(* Logix 5000 project; controller Carpenter_Meter_SCP vendor 1 type 14 code 217 rev 31.11; software revision 31.01 *)

TASK MainTask (continuous, watchdog 500 ms) : First_Scan, Map_Inputs, Alarm_Shutdown, Valve_Control, Station_Overrides, Station_Control, Meter_Skid_Control, Auxiliary_Control, Communication, Map_Outputs, OCC_Comms

MODULES
   Local : vendor 1 type 14 code 217 (5069 0, rev 31.11)
      Carpenter_Meter_FGP : vendor 1 type 14 code 217 (Ethernet 10.131.51.170, rev 31.1, $eaa37dee$ RPI 20 ms, $a3d2e279$ RPI 20 ms)
      MLV_HRF100 : vendor 1 type 14 code 107 (Ethernet 10.171.255.104, rev 31.1)
      Hereford_Meter_SCP : vendor 1 type 14 code 217 (Ethernet 10.131.191.105, rev 31.1)
      MLV_CAR100 : vendor 1 type 14 code 107 (Ethernet 10.171.255.120, rev 31.1)
      Pawnee_EN2T : 1756-EN2T (Ethernet 10.169.41.58, rev 10.1, Output RPI 10 ms)
         PWN : vendor 1 type 14 code 96 (ICP 0, rev 24.1)
      SCP_Main : 5094-AENTR (Ethernet 192.168.2.3, rev 2.1)
         SCP_Main_DOUT1 : 5094-OB16 (5094 3, rev 1.1, StandardDataDriven RPI 5 ms)
         SCP_Main_DIN2 : 5094-IB16 (5094 2, rev 1.1, StandardDataDriven RPI 5 ms)
         SCP_Main_AIN1 : 5094-IF8 (5094 4, rev 1.1, StandardDataDriven RPI 100 ms)
         SCP_Main_DIN1 : 5094-IB16 (5094 1, rev 1.1, StandardDataDriven RPI 5 ms)
      MS8800_SCP_RIO : 5094-AENTR (Ethernet 192.168.2.5, rev 2.1)
         MS8800_SCP_RIO_AIN1 : 5094-IF8 (5094 2, rev 1.1, StandardDataDriven RPI 100 ms)
         MS8800_SCP_RIO_AOUT1 : 5094-OF8 (5094 3, rev 1.1, StandardDataDriven RPI 100 ms)
         MS8800_SCP_RIO_DIN1 : 5094-IB16 (5094 1, rev 1.1, StandardDataDriven RPI 5 ms)
      MS8840_SCP_RIO : 5094-AENTR (Ethernet 192.168.2.7, rev 2.1)
         MS8840_SCP_RIO_DIN1 : 5094-IB16 (5094 1, rev 1.1, StandardDataDriven RPI 5 ms)
         MS8840_SCP_RIO_AOUT1 : 5094-OF8 (5094 3, rev 1.1, StandardDataDriven RPI 100 ms)
         MS8840_SCP_RIO_AIN1 : 5094-IF8 (5094 2, rev 1.1, StandardDataDriven RPI 100 ms)
END_MODULES

TYPE BaseVLVLiquid :   // XV-XXXX
STRUCT
   chg_tmr : TIMER;   // Valve Change Timer
   Cls_CMD : BOOL;   // Valve Close Command
   Cls_Req : BOOL;   // Valve Close Request from OCC
   Close_Req_Tmr : TIMER;   // Valve Close Timer
   Cls_Sts : BOOL;   // Valve on Closed limit switch
   DOT_Cmd : BOOL;   // Valve DOT Command
   DOT_Mode : BOOL;   // Valve in DOT mode
   DOT_req : BOOL;   // Valve DOT Mode Request from OCC
   Expected : BOOL;   // Valve Expected Position. 1=Open
   Failed_OOP : BOOL;   // Valve Failed out of Position
   hmi_Cls_req : BOOL;   // Valve Close Request from HMI
   HMI_DOT_CMD : BOOL;   // Valve DOT Command from HMI
   hmi_DOT_req : BOOL;   // Valve DOT Mode Request from HMI
   hmi_opn_req : BOOL;   // Valve Open Request from HMI
   Last_Pos : BOOL;   // Valve Last Known Position 1=open
   Local : BOOL;   // Valve in Local (From Valve)
   Opn_CMD : BOOL;   // Valve Open Command
   Opn_Req : BOOL;   // Valve Open Request from OCC
   Open_Req_Tmr : TIMER;   // Valve Open Timer
   Opn_Sts : BOOL;   // Valve on Open Limit Switch
   Pos_Fdbk : REAL;   // Valve Percent Open Feedback.
   Startup_bit : BOOL;   // Valve First Scan Bit
   Startup_tmr : TIMER;   // Valve Startup Timer
   Sys_Close_Req : BOOL;   // Valve System PLC Close Request
   Posn_Alm : DiscrAlm;   // Valve Position Alarm
   pos_changed : BOOL;   // Valve Position Changed
   remote : BOOL;   // Valve In Remote(From Valve)
   OOP_alm : DiscrAlm;   // Valve Out of Position alarm
   status : INT;   // Valve Status
   fault : BOOL;   // Valve Faulted
END_STRUCT
END_TYPE

TYPE BasProdCons :   // FGP_SCP Produced and Consumed Tags
STRUCT
   bit : BOOL[64];
   integer : INT[80];
   float : REAL[50];
END_STRUCT
END_TYPE

TYPE BasVlv :
STRUCT
   open_cmd : BOOL;   // open command
   cls_cmd : BOOL;   // close command
   open_stat_1 : BOOL;   // ZSO LS open status 1
   open_stat_2 : BOOL;   // ZSO LS open status 2
   cls_stat_1 : BOOL;   // ZSC LS closed status 1
   cls_stat_2 : BOOL;   // ZSC LS closed status 2
   fail_dir : BOOL;   // valve fail direction 1=FO
   open_intlk : BOOL;   // valve differential pressure open interlock
   hmi_open_req : BOOL;   // HMI open request
   hmi_cls_req : BOOL;   // HMI close request
   open_stat : BOOL;   // Valve overall open status
   cls_stat : BOOL;   // Valve overall closed status
   open_intlk_alm : BOOL;   // valve can't open alarm due to interlock
   dP_act : DINT;   // actual differential pressure across valve
   dP_setpt : DINT;   // maximum differential pressure across valve before opening
   cmd_reset_tmr : TIMER[2];   // hmi command reset timer
END_STRUCT
END_TYPE

TYPE DateTime :
STRUCT
   date_time : DINT[7];   // [0]=year [1]=month [2]=day[3]=hour [4]=min [5]=sec
   day_change : BOOL;   // day has changed
   month_change : BOOL;   // month has changed
   ons : BOOL[32];   // change one shot
END_STRUCT
END_TYPE

TYPE OCC_Analog :
STRUCT
   scaled : REAL;
   inhibit : BOOL;
   malf : BOOL;
END_STRUCT
END_TYPE

TYPE OCC_CV :   // OCC Control Valve
STRUCT
   Pos : REAL;   // Control Valve Position Setpoint to OCC
   PosCmd : REAL;   // Control Valve Position Setpoint to OCC
   Malf : BOOL;   // Control Valve Position Malfunction to OCC
END_STRUCT
END_TYPE

TYPE OCC_SCADA :   // OCC SCADA Tag
STRUCT
   scaled : REAL;   // Analog Scaled Value
   inhibit : BOOL;   // Analog Inhibit
   malf : BOOL;   // Anlog Malfunction
END_STRUCT
END_TYPE

TYPE OCC_Setpoint :   // OCC Setpoint
STRUCT
   active : BOOL;   // Control Active to OCC
   SP : INT;   // Setpoint From OCC
END_STRUCT
END_TYPE

TYPE OCC_Status :
STRUCT
   Status : INT;
END_STRUCT
END_TYPE

TYPE StaCtrl :
STRUCT
   pv : REAL;   // Process Variable
   error_abs : REAL;   // SP-PV error (absolute value)
   error : REAL;   // SP-PV error
   no_act : BOOL;   // No Action Required
   incr_load1 : BOOL;   // increase load step1
   incr_load2 : BOOL;   // increase load step2
   incr_load3 : BOOL;   // increase load step3
   incr_load4 : BOOL;   // increase load step4
   decr_load1 : BOOL;   // decrease load step1
   decr_load2 : BOOL;   // decrease load step2
   decr_load3 : BOOL;   // decrease load step3
   decr_load4 : BOOL;   // decrease load step4
   load_req : BOOL;   // load request
   unld_req : BOOL;   // unload request
   ctrl_perm : BOOL;   // pressure control permissive
   unld_perm : BOOL;   // unload permissive
   active : BOOL;   // active
   disable_ctrl_ww : BOOL;   // disable pressure control from ww
   error_neg : BOOL;   // SP-PV error is negative value
   noact_lvl_ww : INT;   // no action level
   incr_lvl1_ww : INT;   // increase level 1 SP
   incr_lvl2_ww : INT;   // increase level 2 SP
   incr_lvl3_ww : INT;   // increase level 3 SP
   incr_lvl4_ww : INT;   // increase level 4 SP
   decr_lvl1_ww : INT;   // decrease level 1 SP
   decr_lvl2_ww : INT;   // decrease level 2 SP
   decr_lvl3_ww : INT;   // decrease level 3 SP
   decr_lvl4_ww : INT;   // decrease level 4 SP
   incr_lvl1_tmr_pre_ww : DINT;   // increase level 1 timer preset
   incr_lvl2_tmr_pre_ww : DINT;   // increase level 2 timer preset
   incr_lvl3_tmr_pre_ww : DINT;   // increase level 2 timer preset
   incr_lvl4_tmr_pre_ww : DINT;   // increase level 4 timer preset
   decr_lvl1_tmr_pre_ww : DINT;   // decrease level 1 timer preset
   decr_lvl2_tmr_pre_ww : DINT;   // decrease level 2 timer preset
   decr_lvl3_tmr_pre_ww : DINT;   // decrease level 3 timer preset
   decr_lvl4_tmr_pre_ww : DINT;   // decrease level 4 timer preset
   setpoint : INT;   // pressure setpoint
   setpoint_old : INT;   // pressure setpoint old value
   setpoint_ww : INT;   // pressure setpoint from ww
   setpoint_lkw : INT;   // pressure setpoint from gas control
   setpoint_min_ww : INT;   // minimum pressure setpoint ww
   setpoint_max_ww : INT;   // maximum pressure setpoint ww
   priority_lvl : INT;   // pressure control priority level
   ld_unld_tmr : TIMER;   // load unload timer
END_STRUCT
END_TYPE

TYPE StaStartStop :
STRUCT
   step_complete : BOOL[32];   // step satisfied
   output : BOOL[32];   // perform this step
   step_fail : BOOL[32];   // step failure
   hmi_disable_step : BOOL[32];   // disable step from ww
   timer : TIMER[8];   // step timer
   overall_tmr : TIMER;   // overall timer
   wait_reset_tmr : TIMER;   // wait reset timer
   skip_tmr : TIMER;   // skip timer
   abort_tmr : TIMER;   // abort timer
   ww_reset_tmr : TIMER[4];   // ww command reset timer
   complete : BOOL;   // sequence complete
   fail : BOOL;   // sequence failure
   accept : BOOL;   // command accepted
   hmi_alm_clear : BOOL;   // alarm clear from ww
   hmi_wait : BOOL;   // extend wait timer
   hmi_abort : BOOL;   // abort
   hmi_skip : BOOL;   // skip timer
   perm : BOOL;   // permissive
   show_wsa : BOOL;   // show wait skip abort screen
   step_timer_preset : DINT;   // step timer preset
END_STRUCT
END_TYPE

TYPE StaStatus :   // Station Status
STRUCT
   local : BOOL;   // station in local
   hmi_local_req : BOOL;   // request local mode
   remote : BOOL;   // station in remote
   hmi_remote_req : BOOL;   // request remote mode
   standby : BOOL;   // station in standby
   hmi_standby_req : BOOL;   // request standby mode
   attended : BOOL;   // station in attended mode
   unattended : BOOL;   // station in unattended mode
   hmi_attended_req : BOOL;   // request attended mode
   hmi_unattended_req : BOOL;   // request unattended mode
   checkin_req : BOOL;   // operator check-in request
   hmi_checkin_clr : BOOL;   // operator check-in clear from hmi
   online : BOOL;   // station online
   offline : BOOL;   // station offline
   starting : BOOL;   // station start in progress
   stopping : BOOL;   // station stop in progress
   suct_path_alm : BOOL;   // suction path condition alarm
   disch_path_alm : BOOL;   // discharge path condition alarm
   vlv_fail_stop_req : BOOL;   // valve failure station stop request
   vlv_sg_rdy_sta_start : BOOL;   // sidegate valves in position for station start
   no_inhibits_active : BOOL;   // no mainline inhibits active
   no_ovrd_active : BOOL;   // no overrides active
   sta_start_req : BOOL;   // station start request
   hmi_sta_start_req : BOOL;   // station start request from hmi
   sta_stop_req : BOOL;   // station stop request
   hmi_sta_stop_req : BOOL;   // station top request from hmi
   sta_stop_req_occ : BOOL;   // station stop request (indirect) from OCC
   sta_stop_req_alm : BOOL;   // station stop request from active alarm condition
   SP_change_sta : BOOL;   // pressure setpoint change from station HMI
   SP_change_occ : BOOL;   // pressure setpoint change from OCC
   cur_ovrd_priority : INT;   // current station override priority
   min_unit_sta_start_ww : INT;   // minimum number of units for a station start
   min_unit_sta_run_ww : INT;   // minimum number of units for running station
   unit_start_err_sp_ww : INT;   // unit start error setpoint
   unit_stop_err_sp_ww : INT;   // unit stop error setpoint
   online_diff_press_sp : INT;   // differential pressure setpoint across block valve for online status
   sta_ctrl : INT;   // station control status word 0=error 1=ml override active 2=disch press cntrl 3=suct press cntrl 4=no active cntrl
   sta_ovrd : INT;   // station override status word
   sta_mode : INT;   // station mode status word 1=local 2=remote 3=standby
   sta_checkin : INT;   // station checkin status word
   checkin_tmr : TIMER[2];   // operator check-in timer
   cmd_reset_tmr : TIMER[10];   // reset timers for commands and ww hmi interface
   OCC_tmr : TIMER[4];   // OCCcontrol timers
END_STRUCT
END_TYPE

TYPE STRING10 :
STRUCT
   LEN : DINT;
   DATA : SINT[10];
END_STRUCT
END_TYPE

TYPE STRING64 :
STRUCT
   LEN : DINT;
   DATA : SINT[64];
END_STRUCT
END_TYPE

TYPE TGE_AI_UDT :
STRUCT
   AlmActive : BOOL;
   HAlmOnHHAlm : BOOL;
   LAlmOnLLAlm : BOOL;
   InhibActive : BOOL;
   InhibAllEnableCmd : BOOL;
   InhibAllDisableCmd : BOOL;
   AlmMaxPriority : DINT;
   AvgNumberOfSamples : INT;
   AvgTimeBetweenSamples : INT;
   Precision : INT;
   TrendTime : INT;
   Avg : REAL;
   EU : REAL;
   EUMax : REAL;
   EUMin : REAL;
   HHAlmSP : REAL;
   HAlmSP : REAL;
   LAlmSP : REAL;
   LLAlmSP : REAL;
   Raw : REAL;
   RawMax : REAL;
   RawMin : REAL;
   ROC : REAL;
   ROCNegAlmSP : REAL;
   ROCPeriodSP : REAL;
   ROCPosAlmSP : REAL;
   Percent : REAL;
   HHAlm : TGE_Alarm;
   HAlm : TGE_Alarm;
   LAlm : TGE_Alarm;
   LLAlm : TGE_Alarm;
   ROCNegAlm : TGE_Alarm;
   ROCPosAlm : TGE_Alarm;
   MalfAlm : TGE_Alarm;
   Average : TGE_Average;
   Units : STRING10;
   Description : STRING64;
END_STRUCT
END_TYPE

ADD_ON_INSTRUCTION AIScale   (* revision 1.0 *)
VAR_OUTPUT
   scaled : REAL; {visible}   // scaled analog value (EU)
END_VAR
VAR_INPUT
   eng_max_ww : REAL; {visible}   // maximum EU value
   eng_min_ww : REAL; {visible}   // minimum EU value
END_VAR
VAR_OUTPUT
   mA : REAL; {visible}   // adjusted mA signal (calculated)
END_VAR
VAR_INPUT
   max_mA_ww : REAL := 20.0; {visible}   // maximum mA scaling
   min_mA_ww : REAL := 4.0; {visible}   // minimum mA scaling
   physical_Input : REAL; {required}   // analog input signal in counts
END_VAR
VAR
   ma_max_min_diff : DINT; {access None}   // calculated difference max & min mA scaling values
   eng_max_min_diff : DINT; {access None}   // calculated difference max & min EU values
   Timer : TIMER[4]; {access None}   // Alarm Delay Timers
END_VAR

ROUTINE Logic   (* ladder *)
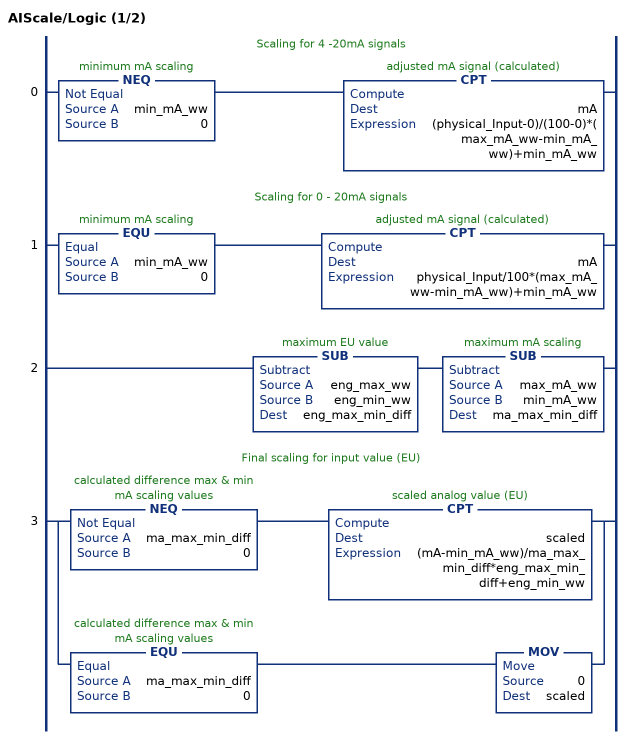
   // Scaling for 4 -20mA signals
   0: NEQ(min_mA_ww,0)CPT(mA,(physical_Input-0)/(100-0)*(max_mA_ww-min_mA_ww)+min_mA_ww);
   // Scaling for 0 - 20mA signals
   1: EQU(min_mA_ww,0)CPT(mA,physical_Input/100*(max_mA_ww-min_mA_ww)+min_mA_ww);
   2: SUB(eng_max_ww,eng_min_ww,eng_max_min_diff)SUB(max_mA_ww,min_mA_ww,ma_max_min_diff);
   // Final scaling for input value (EU)
   3: [NEQ(ma_max_min_diff,0) CPT(scaled,(mA-min_mA_ww)/ma_max_min_diff*eng_max_min_diff+eng_min_ww) ,EQU(ma_max_min_diff,0) MOV(0,scaled) ];
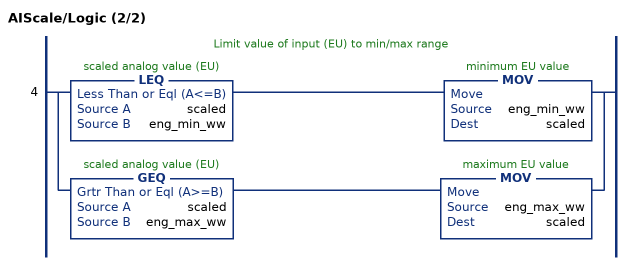
   // Limit value of input (EU) to min/max range
   4: [LEQ(scaled,eng_min_ww) MOV(eng_min_ww,scaled) ,GEQ(scaled,eng_max_ww) MOV(eng_max_ww,scaled) ];
END_ROUTINE
END_ADD_ON_INSTRUCTION

ADD_ON_INSTRUCTION AnalogAlm   (* revision 1.0 *)
VAR_INPUT
   Input : REAL; {access Read Only, required}   // Scaled Analog Value (EU)
   mA : REAL; {access Read Only, required}   // Adjusted mA Signal (Calculated)
   sta_attended : BOOL; {required}   // station attended
END_VAR
VAR_IN_OUT
   alarm_co : BOOL[32]; {required}
END_VAR
VAR_INPUT
   horn_req : BOOL; {required}   // Horn Request
END_VAR
VAR_OUTPUT
   Lo_act : BOOL; {visible}
   Lo_hmi_act : BOOL;
END_VAR
VAR_INPUT
   Lo_horn_ena : BOOL;   // Horn Enable
   Lo_inh_alm : BOOL;
   Lo_inh_ww : BOOL; {visible}
END_VAR
VAR_OUTPUT
   LoLo_act : BOOL; {visible}
   LoLo_hmi_act : BOOL;
END_VAR
VAR_INPUT
   LoLo_horn_ena : BOOL;   // Horn Enable
   LoLo_inh_alm : BOOL;
   LoLo_inh_ww : BOOL; {visible}
END_VAR
VAR_OUTPUT
   Hi_act : BOOL; {visible}
   Hi_hmi_act : BOOL;
END_VAR
VAR_INPUT
   Hi_horn_ena : BOOL;   // Horn Enable
   Hi_inh_alm : BOOL;
   Hi_inh_ww : BOOL; {visible}
END_VAR
VAR_OUTPUT
   HiHi_act : BOOL; {visible}
   HiHi_hmi_act : BOOL;
END_VAR
VAR_INPUT
   HiHi_horn_ena : BOOL;   // Horn Enable
   HiHi_inh_alm : BOOL;
   HiHi_inh_ww : BOOL; {visible}
END_VAR
VAR_OUTPUT
   Malf_act : BOOL; {visible}
   Malf_hmi_act : BOOL;
END_VAR
VAR_INPUT
   Malf_inh_alm : BOOL;
   Malf_inh_ww : BOOL;
END_VAR
VAR_OUTPUT
   Malf_immed : BOOL;   // immediate malfunction flag
END_VAR
VAR_INPUT
   Lo_setpt : REAL; {visible}
   LoLo_setpt : REAL; {visible}
   Hi_setpt : REAL; {visible}
   HiHi_setpt : REAL; {visible}
   Lo_tmr_pre : DINT; {visible}
   Lo_tmr_pre_recur : DINT;
   LoLo_tmr_pre : DINT; {visible}
   LoLo_tmr_pre_recur : DINT;
   Hi_tmr_pre : DINT; {visible}
   Hi_tmr_pre_recur : DINT;
   HiHi_tmr_pre : DINT; {visible}
   HiHi_tmr_pre_recur : DINT;
   Malf_tmr_pre : DINT;
   Malf_tmr_pre_recur : DINT;
   Lo_co_type : INT;   // Lo Alarm Callout Type
   LoLo_co_type : INT;   // LoLo Alarm Callout Type
   Hi_co_type : INT;   // Hi Alarm Callout Type
   HiHi_co_type : INT;   // HiHi Alarm Callout Type
   Malf_co_type : INT;   // Malf Alarm Callout Type
END_VAR
VAR
   alarm_ons : BOOL[32]; {access None}
   timer : TIMER[10]; {access None}
        [0]   // malf active timer
        [1]   // malf recurring timer
        [2]   // lo active timer
        [3]   // lo recurring timer
        [4]   // lolo active timer
        [5]   // lolo recurring timer
        [6]   // hi active timer
        [7]   // hi recurring timer
        [8]   // hihi active timer
        [9]   // hihi recurring timer
   co_index : INT; {access None}
END_VAR

ROUTINE Logic   (* ladder *)
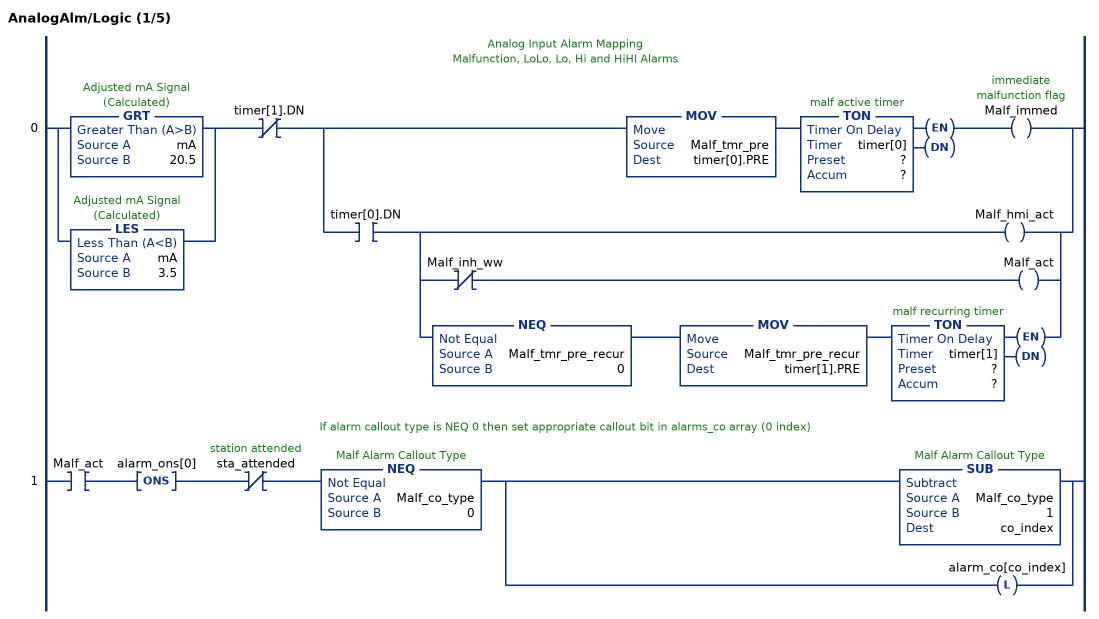
   // Analog Input Alarm Mapping
   // Malfunction, LoLo, Lo, Hi and HiHI Alarms
   0: [GRT(mA,20.5) ,LES(mA,3.5) ]XIO(timer[1].DN)[MOV(Malf_tmr_pre,timer[0].PRE) TON(timer[0],?,?) OTE(Malf_immed) ,XIC(timer[0].DN) [[OTE(Malf_hmi_act) ,XIO(Malf_inh_ww) OTE(Malf_act) ] ,NEQ(Malf_tmr_pre_recur,0) MOV(Malf_tmr_pre_recur,timer[1].PRE) TON(timer[1],?,?) ] ];
   // If alarm callout type is NEQ 0 then set appropriate callout bit in alarms_co array (0 index)
   1: XIC(Malf_act)ONS(alarm_ons[0])XIO(sta_attended)NEQ(Malf_co_type,0)[SUB(Malf_co_type,1,co_index) ,OTL(alarm_co[co_index]) ];
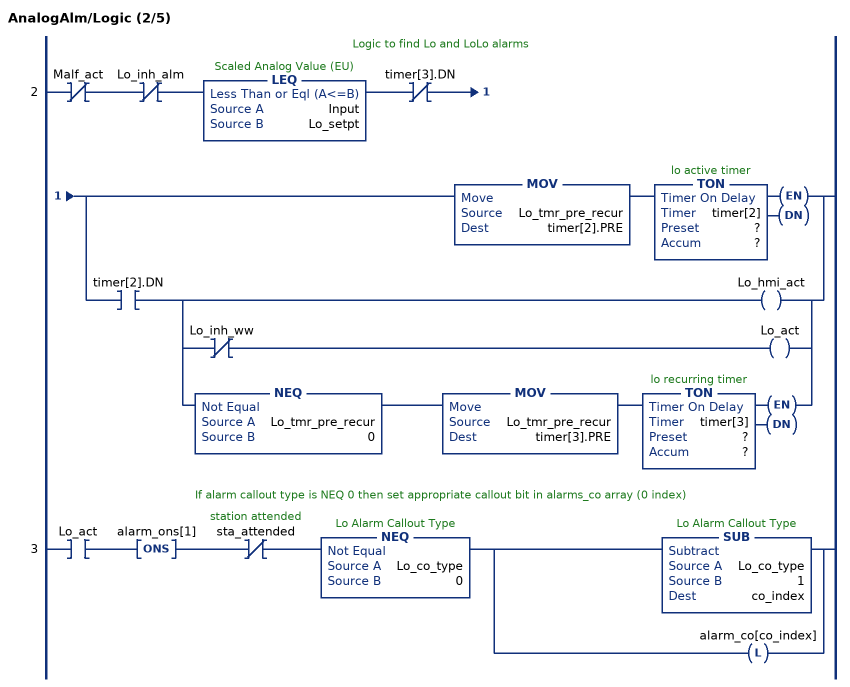
   // Logic to find Lo and LoLo alarms
   2: XIO(Malf_act)XIO(Lo_inh_alm)LEQ(Input,Lo_setpt)XIO(timer[3].DN)[MOV(Lo_tmr_pre_recur,timer[2].PRE) TON(timer[2],?,?) ,XIC(timer[2].DN) [[OTE(Lo_hmi_act) ,XIO(Lo_inh_ww) OTE(Lo_act) ] ,NEQ(Lo_tmr_pre_recur,0) MOV(Lo_tmr_pre_recur,timer[3].PRE) TON(timer[3],?,?) ] ];
   // If alarm callout type is NEQ 0 then set appropriate callout bit in alarms_co array (0 index)
   3: XIC(Lo_act)ONS(alarm_ons[1])XIO(sta_attended)NEQ(Lo_co_type,0)[SUB(Lo_co_type,1,co_index) ,OTL(alarm_co[co_index]) ];
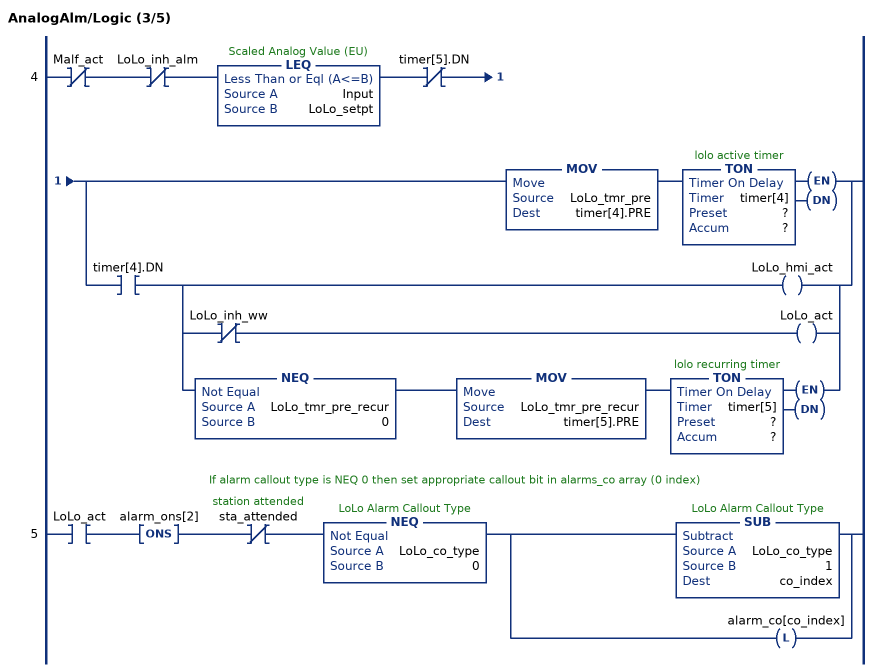
   4: XIO(Malf_act)XIO(LoLo_inh_alm)LEQ(Input,LoLo_setpt)XIO(timer[5].DN)[MOV(LoLo_tmr_pre,timer[4].PRE) TON(timer[4],?,?) ,XIC(timer[4].DN) [[OTE(LoLo_hmi_act) ,XIO(LoLo_inh_ww) OTE(LoLo_act) ] ,NEQ(LoLo_tmr_pre_recur,0) MOV(LoLo_tmr_pre_recur,timer[5].PRE) TON(timer[5],?,?) ] ];
   // If alarm callout type is NEQ 0 then set appropriate callout bit in alarms_co array (0 index)
   5: XIC(LoLo_act)ONS(alarm_ons[2])XIO(sta_attended)NEQ(LoLo_co_type,0)[SUB(LoLo_co_type,1,co_index) ,OTL(alarm_co[co_index]) ];
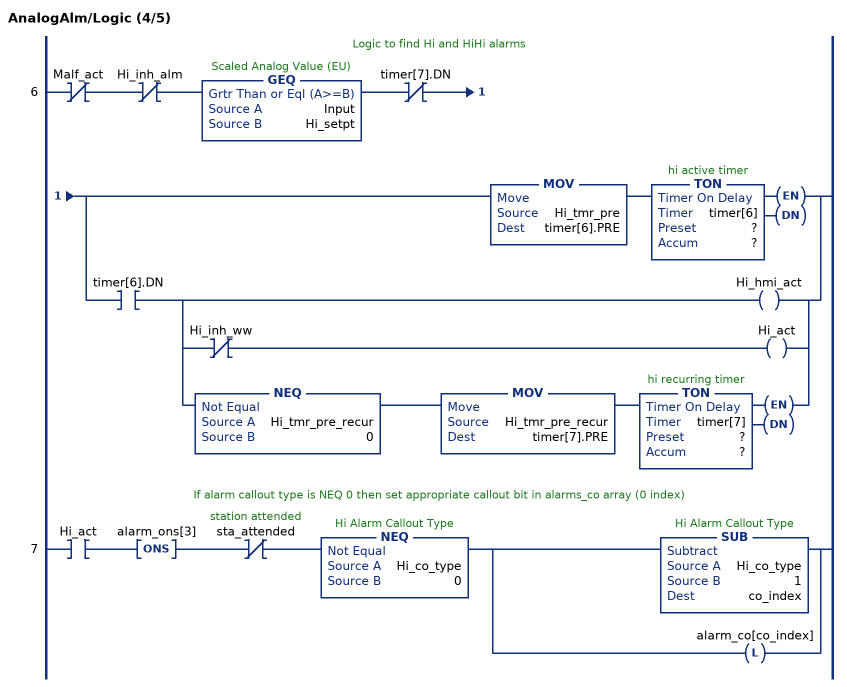
   // Logic to find Hi and HiHi alarms
   6: XIO(Malf_act)XIO(Hi_inh_alm)GEQ(Input,Hi_setpt)XIO(timer[7].DN)[MOV(Hi_tmr_pre,timer[6].PRE) TON(timer[6],?,?) ,XIC(timer[6].DN) [[OTE(Hi_hmi_act) ,XIO(Hi_inh_ww) OTE(Hi_act) ] ,NEQ(Hi_tmr_pre_recur,0) MOV(Hi_tmr_pre_recur,timer[7].PRE) TON(timer[7],?,?) ] ];
   // If alarm callout type is NEQ 0 then set appropriate callout bit in alarms_co array (0 index)
   7: XIC(Hi_act)ONS(alarm_ons[3])XIO(sta_attended)NEQ(Hi_co_type,0)[SUB(Hi_co_type,1,co_index) ,OTL(alarm_co[co_index]) ];
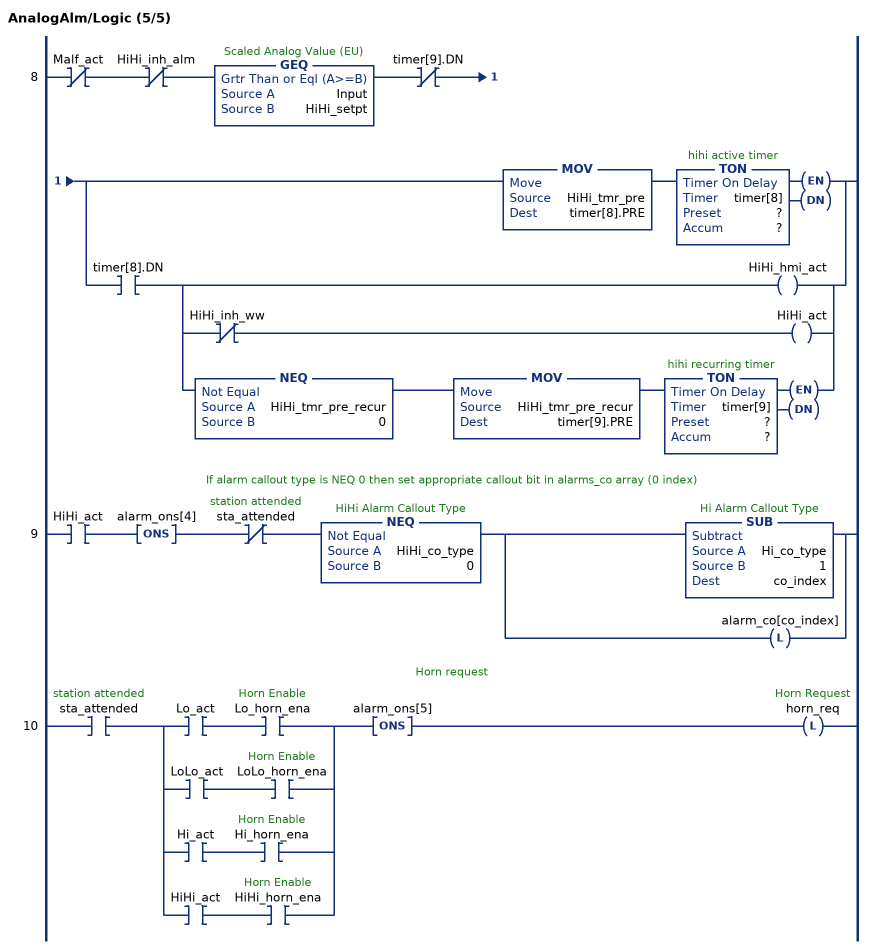
   8: XIO(Malf_act)XIO(HiHi_inh_alm)GEQ(Input,HiHi_setpt)XIO(timer[9].DN)[MOV(HiHi_tmr_pre,timer[8].PRE) TON(timer[8],?,?) ,XIC(timer[8].DN) [[OTE(HiHi_hmi_act) ,XIO(HiHi_inh_ww) OTE(HiHi_act) ] ,NEQ(HiHi_tmr_pre_recur,0) MOV(HiHi_tmr_pre_recur,timer[9].PRE) TON(timer[9],?,?) ] ];
   // If alarm callout type is NEQ 0 then set appropriate callout bit in alarms_co array (0 index)
   9: XIC(HiHi_act)ONS(alarm_ons[4])XIO(sta_attended)NEQ(HiHi_co_type,0)[SUB(Hi_co_type,1,co_index) ,OTL(alarm_co[co_index]) ];
   // Horn request
   10: XIC(sta_attended)[XIC(Lo_act) XIC(Lo_horn_ena) ,XIC(LoLo_act) XIC(LoLo_horn_ena) ,XIC(Hi_act) XIC(Hi_horn_ena) ,XIC(HiHi_act) XIC(HiHi_horn_ena) ]ONS(alarm_ons[5])OTL(horn_req);
END_ROUTINE
END_ADD_ON_INSTRUCTION

ADD_ON_INSTRUCTION AOScale   (* revision 1.0 *)
VAR_OUTPUT
   scaled_output : REAL; {required}   // scaled analog signal in counts
END_VAR
VAR_INPUT
   eng_max_ww : REAL; {visible}   // maximum EU value
   eng_min_ww : REAL; {visible}   // minimum EU value
END_VAR
VAR_OUTPUT
   mA : REAL; {visible}   // adjusted mA signal (calculated)
END_VAR
VAR_INPUT
   max_mA_ww : REAL; {visible}   // maximum mA scaling
   min_mA_ww : REAL; {visible}   // minimum mA scaling
   cmd_input : DINT; {required}   // scaled command input
END_VAR
VAR
   ma_max_min_diff : DINT; {access None}   // calculated difference max & min mA scaling values
   eng_max_min_diff : DINT; {access None}   // calculated difference max & min EU values
   Timer : TIMER[4]; {access None}   // Alarm Delay Timers
END_VAR

ROUTINE Logic   (* ladder *)
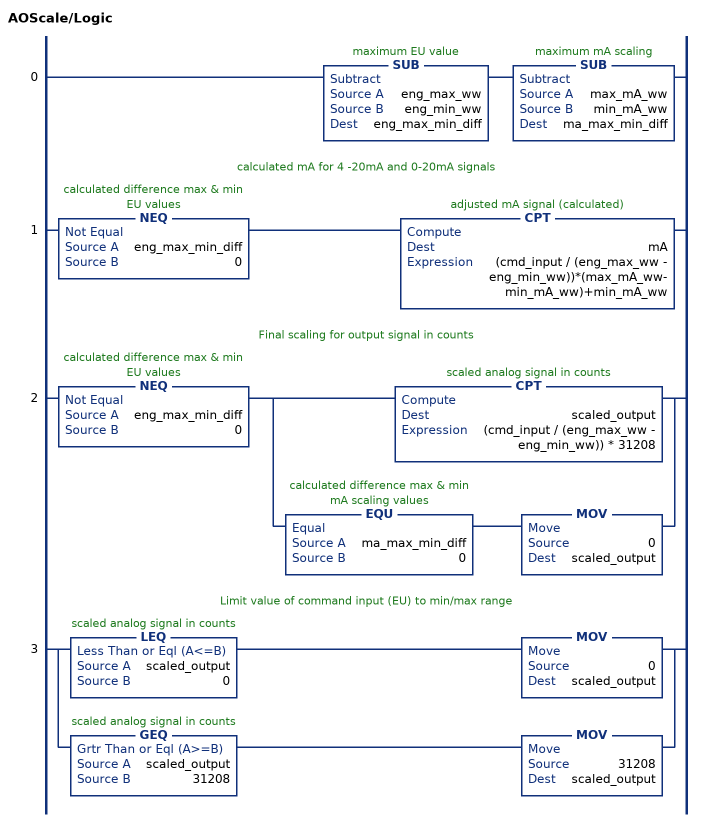
   0: SUB(eng_max_ww,eng_min_ww,eng_max_min_diff)SUB(max_mA_ww,min_mA_ww,ma_max_min_diff);
   // calculated mA for 4 -20mA and 0-20mA signals
   1: NEQ(eng_max_min_diff,0)CPT(mA,(cmd_input / (eng_max_ww - eng_min_ww))*(max_mA_ww-min_mA_ww)+min_mA_ww);
   // Final scaling for output signal in counts
   2: NEQ(eng_max_min_diff,0)[CPT(scaled_output,(cmd_input / (eng_max_ww - eng_min_ww)) * 31208) ,EQU(ma_max_min_diff,0) MOV(0,scaled_output) ];
   // Limit value of command input (EU) to min/max range
   3: [LEQ(scaled_output,0) MOV(0,scaled_output) ,GEQ(scaled_output,31208) MOV(31208,scaled_output) ];
END_ROUTINE
END_ADD_ON_INSTRUCTION

ADD_ON_INSTRUCTION DiscrAlm   (* revision 1.0 *)
// Discrete Alarm AOI
VAR_INPUT
   input : BOOL;   // discrete alarm input signal
END_VAR
VAR_IN_OUT
   alarm_co : BOOL[32]; {required}
END_VAR
VAR_INPUT
   horn_req : BOOL; {required}   // horn request
   sta_attended : BOOL; {required}   // station attended
END_VAR
VAR_OUTPUT
   alm_act : BOOL; {visible}
   alm_hmi_act : BOOL;
END_VAR
VAR_INPUT
   inh_alm : BOOL;   // used as master inhibit for entire alarm
END_VAR
VAR_OUTPUT
   horn_enable : BOOL; {visible}   // enable alarm to sound FGP building horns
END_VAR
VAR_INPUT
   alm_inh_ww : BOOL; {visible}
   alm_tmr_pre : DINT; {visible}
   alm_tmr_pre_recur : DINT;
   co_type : INT;   // active alarm callout type
END_VAR
VAR
   alarm_ons : BOOL[32]; {access None}
   timer : TIMER[2]; {access None}
        [0]   // alarm active timer
        [1]   // alarm recurring timer
   co_index : INT; {access None}
END_VAR

ROUTINE Logic   (* ladder *)
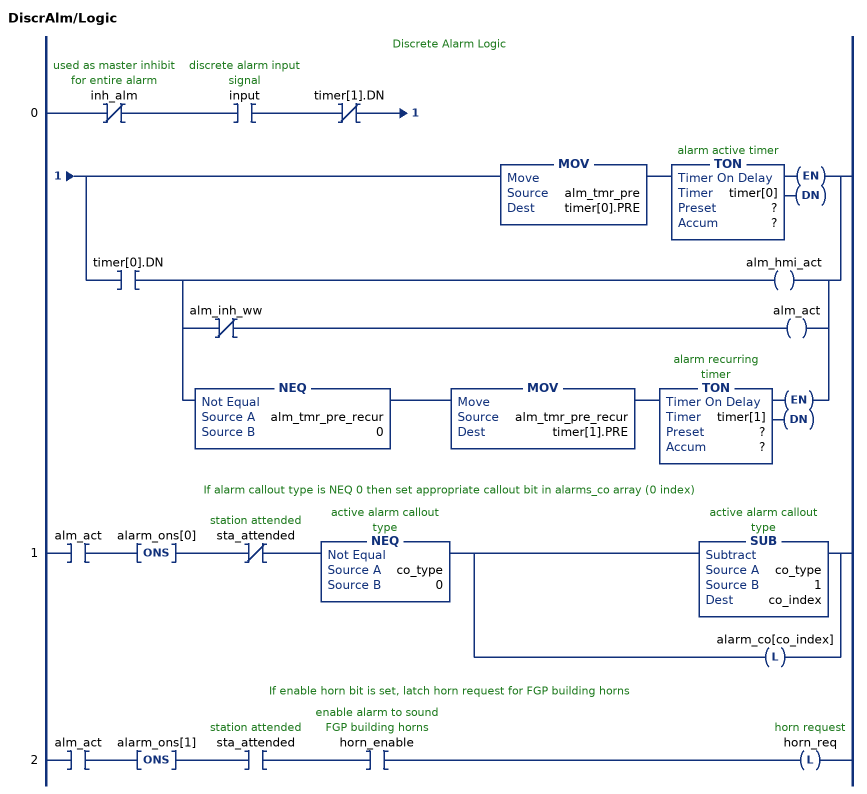
   // Discrete Alarm Logic
   0: XIO(inh_alm)XIC(input)XIO(timer[1].DN)[MOV(alm_tmr_pre,timer[0].PRE) TON(timer[0],?,?) ,XIC(timer[0].DN) [[OTE(alm_hmi_act) ,XIO(alm_inh_ww) OTE(alm_act) ] ,NEQ(alm_tmr_pre_recur,0) MOV(alm_tmr_pre_recur,timer[1].PRE) TON(timer[1],?,?) ] ];
   // If alarm callout type is NEQ 0 then set appropriate callout bit in alarms_co array (0 index)
   1: XIC(alm_act)ONS(alarm_ons[0])XIO(sta_attended)NEQ(co_type,0)[SUB(co_type,1,co_index) ,OTL(alarm_co[co_index]) ];
   // If enable horn bit is set, latch horn request for FGP building horns
   2: XIC(alm_act)ONS(alarm_ons[1])XIC(sta_attended)XIC(horn_enable)OTL(horn_req);
END_ROUTINE
END_ADD_ON_INSTRUCTION

ADD_ON_INSTRUCTION IntrusionAlm   (* revision 1.0 *)
VAR_IN_OUT
   alarm_co : BOOL[32]; {required}
END_VAR
VAR_INPUT
   sta_attended : BOOL; {required}   // Station Attended
END_VAR
VAR_OUTPUT
   alm_act : BOOL; {visible}
   alm_hmi_act : BOOL;
END_VAR
VAR_INPUT
   inh_alm : BOOL;
   alm_inh_ww : BOOL; {visible}
   intrusion_act : BOOL; {required}   // Intrusion alarm system active
   alm_tmr_pre : DINT; {visible}
   alm_tmr_pre_recur : DINT;
   co_type : INT;   // Hi Alarm Callout Type
   sw_input : INT;   // b0-7 = bldg instrusion switch b15 = deactive HS
   sw_alm_out : INT;   // b0-7 = bldg intrusion switch alarm
END_VAR
VAR
   alarm_ons : BOOL[32]; {access None}
   timer : TIMER[3]; {access None}
        [0]   // alarm active timer
        [1]   // alarm recurring timer
   co_index : INT; {access None}
END_VAR

ROUTINE Logic   (* ladder *)
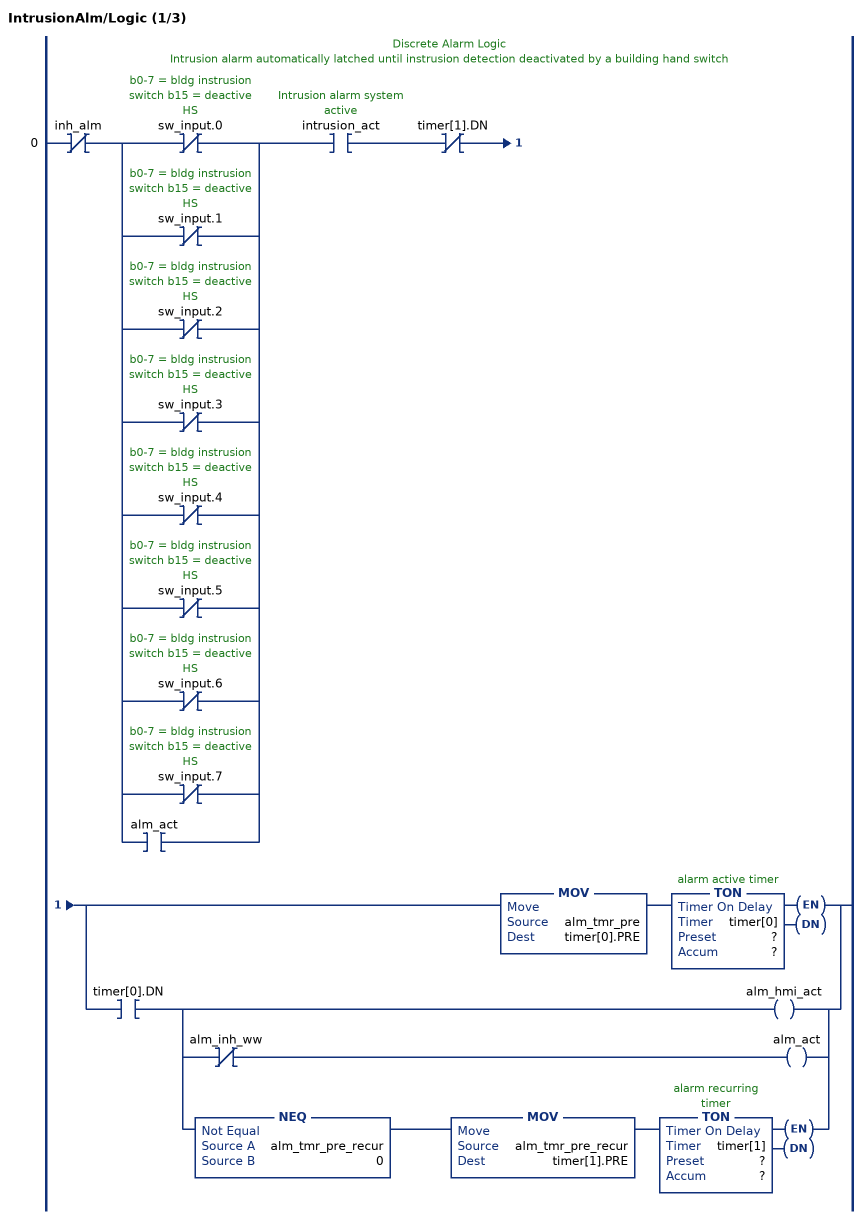
   // Discrete Alarm Logic
   // Intrusion alarm automatically latched until instrusion detection deactivated by a building hand switch
   0: XIO(inh_alm)[XIO(sw_input.0) ,XIO(sw_input.1) ,XIO(sw_input.2) ,XIO(sw_input.3) ,XIO(sw_input.4) ,XIO(sw_input.5) ,XIO(sw_input.6) ,XIO(sw_input.7) ,XIC(alm_act) ]XIC(intrusion_act)XIO(timer[1].DN)[MOV(alm_tmr_pre,timer[0].PRE) TON(timer[0],?,?) ,XIC(timer[0].DN) [[OTE(alm_hmi_act) ,XIO(alm_inh_ww) OTE(alm_act) ] ,NEQ(alm_tmr_pre_recur,0) MOV(alm_tmr_pre_recur,timer[1].PRE) TON(timer[1],?,?) ] ];
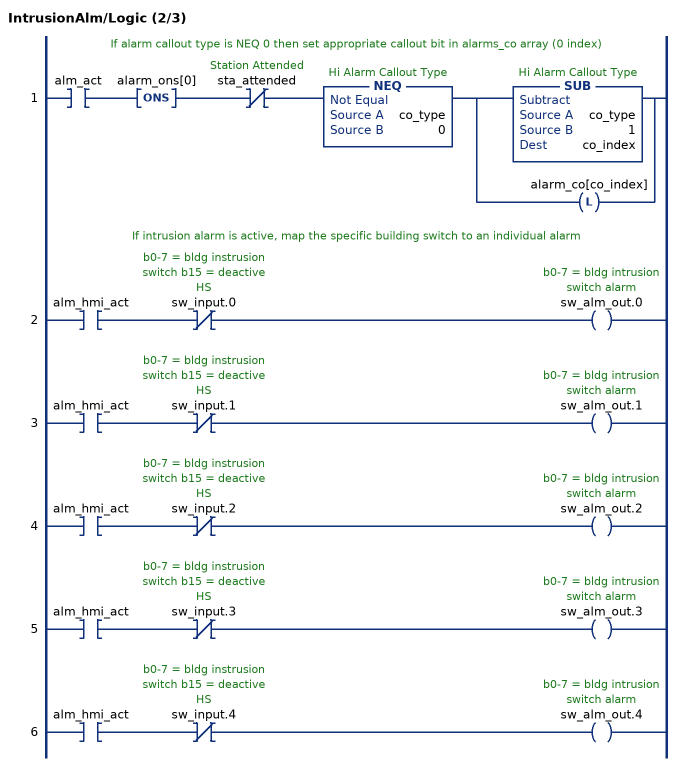
   // If alarm callout type is NEQ 0 then set appropriate callout bit in alarms_co array (0 index)
   1: XIC(alm_act)ONS(alarm_ons[0])XIO(sta_attended)NEQ(co_type,0)[SUB(co_type,1,co_index) ,OTL(alarm_co[co_index]) ];
   // If intrusion alarm is active, map the specific building switch to an individual alarm
   2: XIC(alm_hmi_act)XIO(sw_input.0)OTE(sw_alm_out.0);
   3: XIC(alm_hmi_act)XIO(sw_input.1)OTE(sw_alm_out.1);
   4: XIC(alm_hmi_act)XIO(sw_input.2)OTE(sw_alm_out.2);
   5: XIC(alm_hmi_act)XIO(sw_input.3)OTE(sw_alm_out.3);
   6: XIC(alm_hmi_act)XIO(sw_input.4)OTE(sw_alm_out.4);
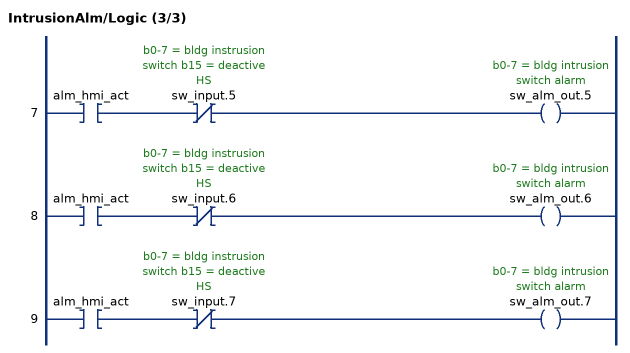
   7: XIC(alm_hmi_act)XIO(sw_input.5)OTE(sw_alm_out.5);
   8: XIC(alm_hmi_act)XIO(sw_input.6)OTE(sw_alm_out.6);
   9: XIC(alm_hmi_act)XIO(sw_input.7)OTE(sw_alm_out.7);
END_ROUTINE
END_ADD_ON_INSTRUCTION

ADD_ON_INSTRUCTION LocalDateTime   (* revision 1.0 *)
VAR_OUTPUT
   Year : ALIAS FOR WallClockValues[0]; {access Read Only, visible}   // Year [YYYY]
   Month : ALIAS FOR WallClockValues[1]; {access Read Only, visible}   // Month (1...12)
   Day : ALIAS FOR WallClockValues[2]; {access Read Only, visible}   // Day (1...31)
   Hour : ALIAS FOR WallClockValues[3]; {access Read Only, visible}   // Hour (0...23)
   Minute : ALIAS FOR WallClockValues[4]; {access Read Only, visible}   // Minute (0...59)
   Second : ALIAS FOR WallClockValues[5]; {access Read Only, visible}   // Seconds (0...59)
   mSec : DINT; {access Read Only, visible}   // Milliseconds (uSec/1000)
   uSec : ALIAS FOR WallClockValues[6]; {access Read Only, visible}   // Microseconds (0...999,999)
   HhMmSs : DINT; {access Read Only, visible}   // HHMMSS Format
END_VAR
VAR
   WallClockValues : DINT[7]; {access Read Only}   // Wall Clock:
        [0]   // Year [YYYY]
        [1]   // Month (1...12)
        [2]   // Day (1...31)
        [3]   // Hour (0...23)
        [4]   // Minute (0...59)
        [5]   // Seconds (0...59)
        [6]   // Microseconds (0...999,999)
END_VAR

ROUTINE Logic   (* ladder *)
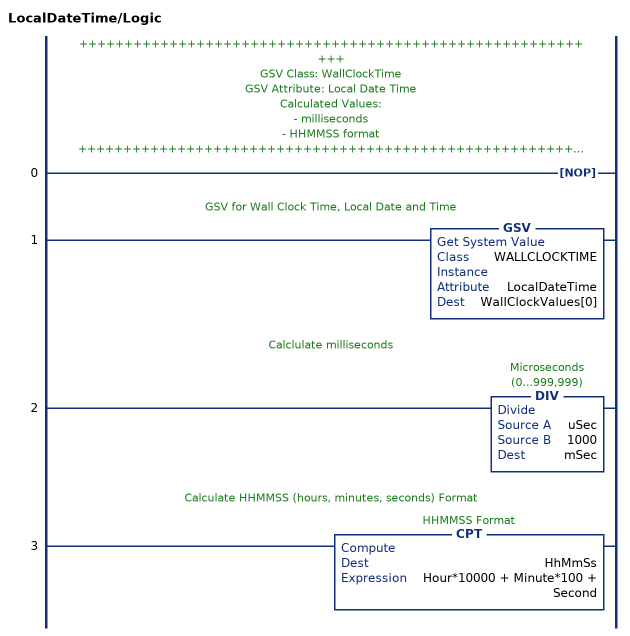
   // +++++++++++++++++++++++++++++++++++++++++++++++++++++++++++
   // GSV Class: WallClockTime
   // GSV Attribute: Local Date Time
   // Calculated Values:
   // - milliseconds
   // - HHMMSS format
   // +++++++++++++++++++++++++++++++++++++++++++++++++++++++++++
   0: NOP();
   // GSV for Wall Clock Time, Local Date and Time
   1: GSV(WALLCLOCKTIME,,LocalDateTime,WallClockValues[0]);
   // Calclulate milliseconds
   2: DIV(uSec,1000,mSec);
   // Calculate HHMMSS (hours, minutes, seconds) Format
   3: CPT(HhMmSs,Hour*10000 + Minute*100 + Second);
END_ROUTINE
END_ADD_ON_INSTRUCTION

ADD_ON_INSTRUCTION Override   (* revision 1.0 *)
VAR_INPUT
   pv : REAL; {visible}
   pv_abs_val : REAL;
   ovrd_request : BOOL;   // override request
END_VAR
VAR_OUTPUT
   highest_type : BOOL; {visible}   // override has highest type
END_VAR
VAR_INPUT
   hmi_alm_clear : BOOL;   // override alarm clear
END_VAR
VAR_OUTPUT
   active : BOOL; {visible}   // override active
   inhibit : BOOL; {visible}   // inhibit active
   hmi_unload_1 : BOOL; {visible}   // unload 1 active hmi
END_VAR
VAR_INPUT
   unload_1 : BOOL;   // unload 1 active
   unload_1_pulse : BOOL;
END_VAR
VAR_OUTPUT
   hmi_unload_all : BOOL; {visible}   // unload all active hmi
END_VAR
VAR_INPUT
   unload_all : BOOL;   // unload all active
   unload_all_pulse : BOOL;
END_VAR
VAR_OUTPUT
   hmi_stop_1 : BOOL; {visible}   // stop 1 active hmi
END_VAR
VAR_INPUT
   stop_1 : BOOL;   // stop 1 active
   stop_1_pulse : BOOL;
END_VAR
VAR_OUTPUT
   jmp_to_stop : BOOL; {visible}   // jump to stop flag
   sta_stop : BOOL; {visible}   // station stop active
END_VAR
VAR_INPUT
   ovrd_type : INT;   // override type
   inh_sp : REAL; {visible}   // inhibit setpoint
   inh_sp_clr : REAL;   // inhibit clear setpoint
   unld1_sp : REAL; {visible}   // unload 1 setpoint
   unld1_sp_clr : REAL;   // unload 1 clear setpoint
   unldall_sp : REAL; {visible}   // unload all setpoint
   unldall_sp_clr : REAL;   // unload all clear setpoint
   stop1_sp : REAL; {visible}   // stop 1 setpoint
   stop1_sp_clr : REAL;   // stop 1 clear setpoint
   sta_stop_sp : REAL; {visible}   // station stop setpoint
   priority_ww : INT;   // override priority level
   unld_1_tmr_pre : DINT;   // unload 1 inverval timer preset
   unload_all_tmr_pre : DINT;   // unload all interval timer preset
   stop_tmr_pre : DINT;   // unit stop inverval timer preset
   unload_dly_stop_tmr_pre : DINT;   // overall max time to station stop timer preset
   inh_clr_tmr_pre : DINT;   // inhibit clear delay timer preset
   unit_running : BOOL; {required}   // at least one unit running
   unit_remote : BOOL; {required}   // at least one unit in remote
   unit_min_load : BOOL; {required}   // units at min load delay done
   standby : BOOL; {required}   // Station in Standby
END_VAR
VAR
   tmr : TIMER[8] := ([0].PRE := 2000, [5].PRE := 2000, [6].PRE := 2000); {access None}
        [0]   // inhibit clear delay timer
        [1]   // unload 1 inverval timer
        [2]   // unload all interval timer
        [3]   // stop 1 interval timer
        [4]   // unload delay to stop timer
        [5]   // alarm clear timer
        [6]   // jmp to stop flag tmr
END_VAR

ROUTINE Logic   (* ladder *)
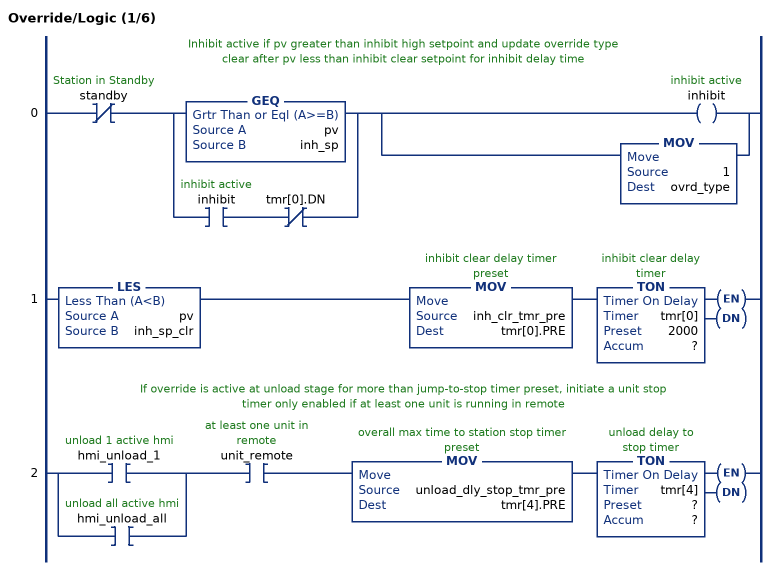
   // Inhibit active if pv greater than inhibit high setpoint and update override type
   // clear after pv less than inhibit clear setpoint for inhibit delay time
   0: XIO(standby)[GEQ(pv,inh_sp) ,XIC(inhibit) XIO(tmr[0].DN) ][OTE(inhibit) ,MOV(1,ovrd_type) ];
   1: LES(pv,inh_sp_clr)MOV(inh_clr_tmr_pre,tmr[0].PRE)TON(tmr[0],?,?);
   // If override is active at unload stage for more than jump-to-stop timer preset, initiate a unit stop
   // timer only enabled if at least one unit is running in remote
   2: [XIC(hmi_unload_1) ,XIC(hmi_unload_all) ]XIC(unit_remote)MOV(unload_dly_stop_tmr_pre,tmr[4].PRE)TON(tmr[4],?,?);
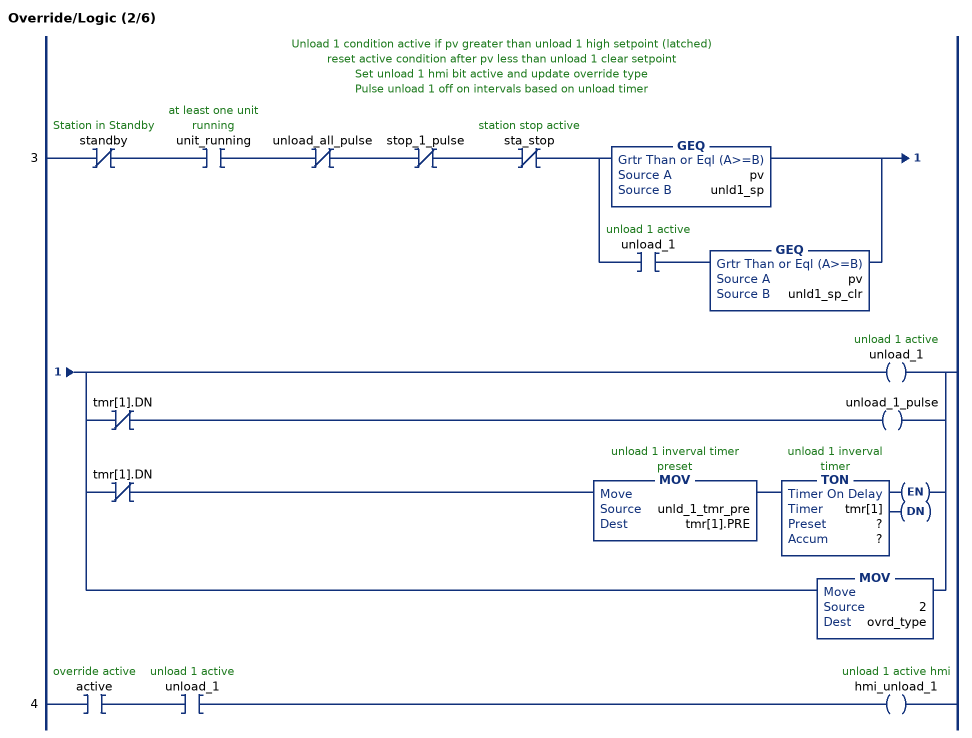
   // Unload 1 condition active if pv greater than unload 1 high setpoint (latched)
   // reset active condition after pv less than unload 1 clear setpoint
   // Set unload 1 hmi bit active and update override type
   // Pulse unload 1 off on intervals based on unload timer
   3: XIO(standby)XIC(unit_running)XIO(unload_all_pulse)XIO(stop_1_pulse)XIO(sta_stop)[GEQ(pv,unld1_sp) ,XIC(unload_1) GEQ(pv,unld1_sp_clr) ][OTE(unload_1) ,XIO(tmr[1].DN) OTE(unload_1_pulse) ,XIO(tmr[1].DN) MOV(unld_1_tmr_pre,tmr[1].PRE) TON(tmr[1],?,?) ,MOV(2,ovrd_type) ];
   4: XIC(active)XIC(unload_1)OTE(hmi_unload_1);
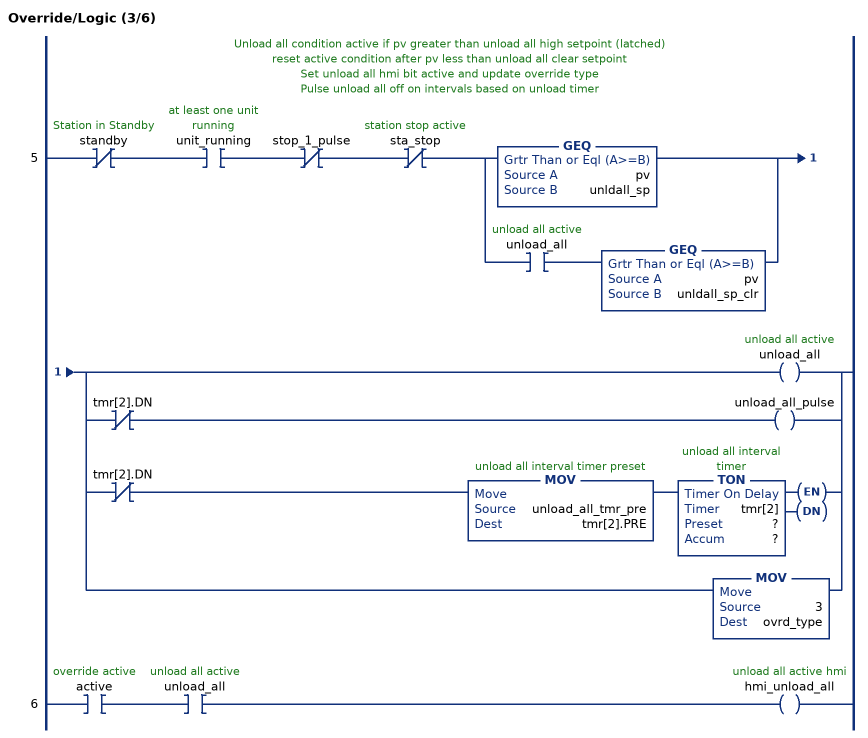
   // Unload all condition active if pv greater than unload all high setpoint (latched)
   // reset active condition after pv less than unload all clear setpoint
   // Set unload all hmi bit active and update override type
   // Pulse unload all off on intervals based on unload timer
   5: XIO(standby)XIC(unit_running)XIO(stop_1_pulse)XIO(sta_stop)[GEQ(pv,unldall_sp) ,XIC(unload_all) GEQ(pv,unldall_sp_clr) ][OTE(unload_all) ,XIO(tmr[2].DN) OTE(unload_all_pulse) ,XIO(tmr[2].DN) MOV(unload_all_tmr_pre,tmr[2].PRE) TON(tmr[2],?,?) ,MOV(3,ovrd_type) ];
   6: XIC(active)XIC(unload_all)OTE(hmi_unload_all);
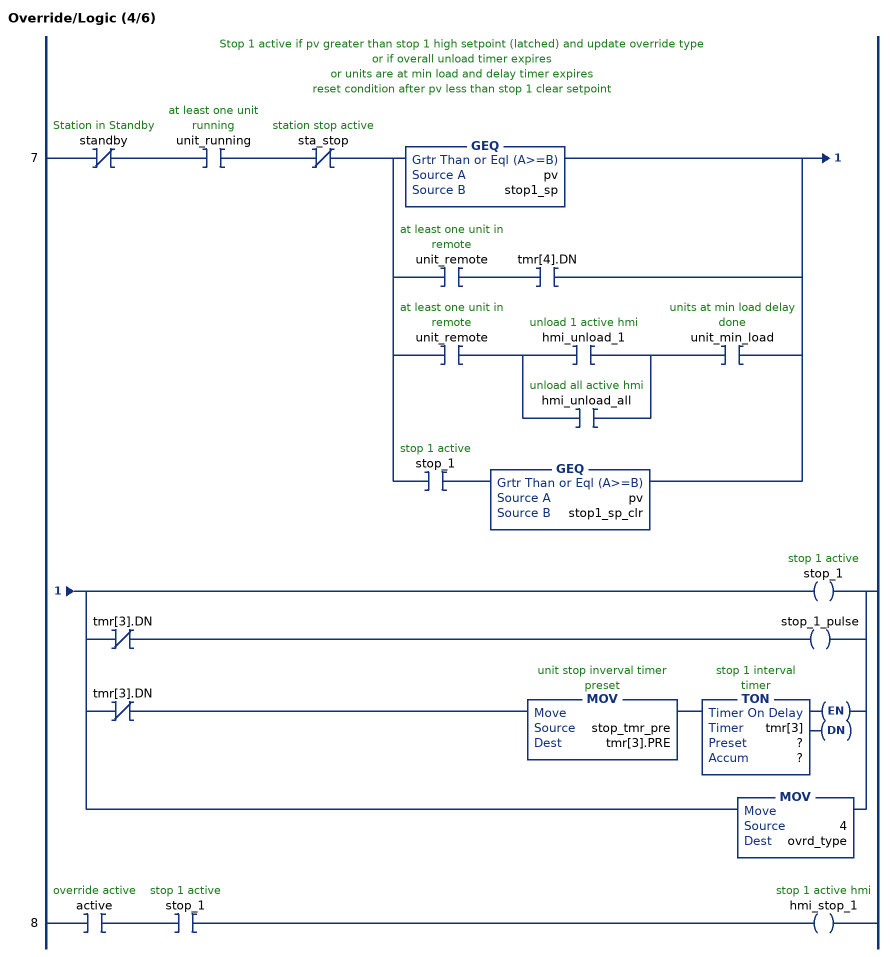
   // Stop 1 active if pv greater than stop 1 high setpoint (latched) and update override type
   // or if overall unload timer expires
   // or units are at min load and delay timer expires
   // reset condition after pv less than stop 1 clear setpoint
   7: XIO(standby)XIC(unit_running)XIO(sta_stop)[GEQ(pv,stop1_sp) ,XIC(unit_remote) XIC(tmr[4].DN) ,XIC(unit_remote) [XIC(hmi_unload_1) ,XIC(hmi_unload_all) ] XIC(unit_min_load) ,XIC(stop_1) GEQ(pv,stop1_sp_clr) ][OTE(stop_1) ,XIO(tmr[3].DN) OTE(stop_1_pulse) ,XIO(tmr[3].DN) MOV(stop_tmr_pre,tmr[3].PRE) TON(tmr[3],?,?) ,MOV(4,ovrd_type) ];
   8: XIC(active)XIC(stop_1)OTE(hmi_stop_1);
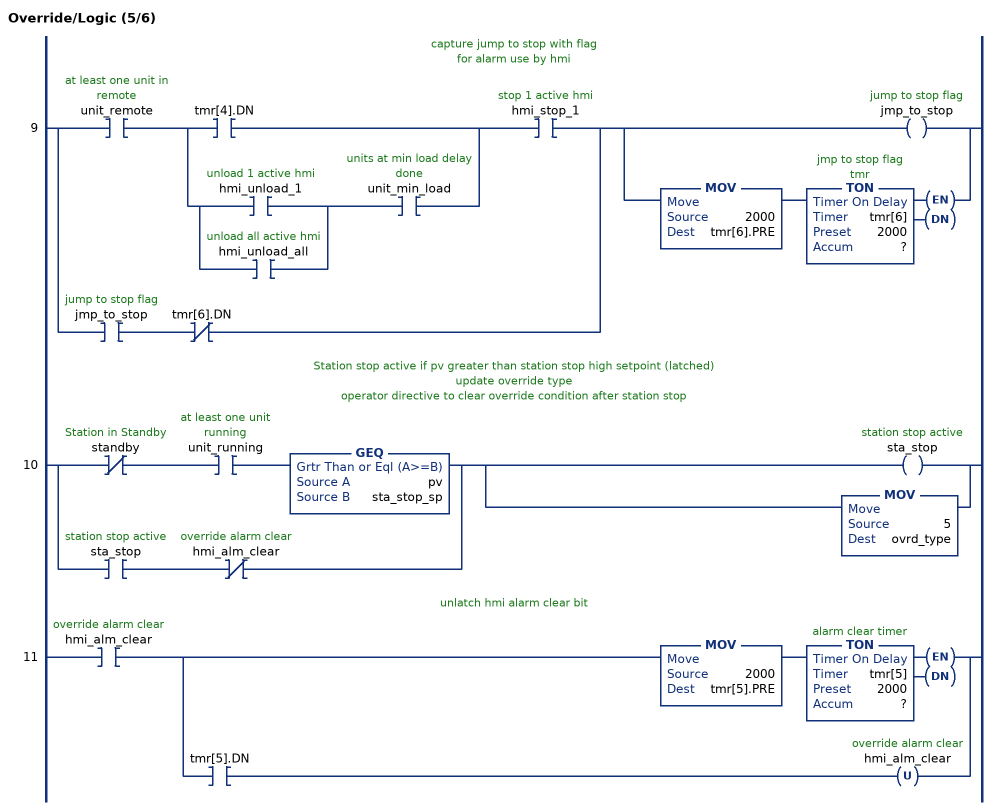
   // capture jump to stop with flag
   // for alarm use by hmi
   9: [XIC(unit_remote) [XIC(tmr[4].DN) ,[XIC(hmi_unload_1) ,XIC(hmi_unload_all) ] XIC(unit_min_load) ] XIC(hmi_stop_1) ,XIC(jmp_to_stop) XIO(tmr[6].DN) ][OTE(jmp_to_stop) ,MOV(2000,tmr[6].PRE) TON(tmr[6],?,?) ];
   // Station stop active if pv greater than station stop high setpoint (latched)
   // update override type
   // operator directive to clear override condition after station stop
   10: [XIO(standby) XIC(unit_running) GEQ(pv,sta_stop_sp) ,XIC(sta_stop) XIO(hmi_alm_clear) ][OTE(sta_stop) ,MOV(5,ovrd_type) ];
   // unlatch hmi alarm clear bit
   11: XIC(hmi_alm_clear)[MOV(2000,tmr[5].PRE) TON(tmr[5],?,?) ,XIC(tmr[5].DN) OTU(hmi_alm_clear) ];
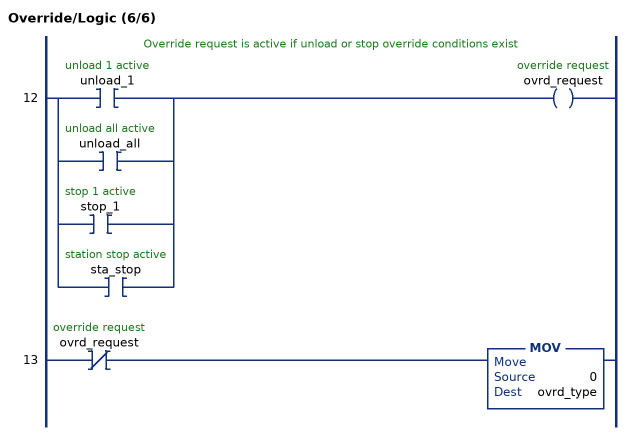
   // Override request is active if unload or stop override conditions exist
   12: [XIC(unload_1) ,XIC(unload_all) ,XIC(stop_1) ,XIC(sta_stop) ]OTE(ovrd_request);
   13: XIO(ovrd_request)MOV(0,ovrd_type);
END_ROUTINE
END_ADD_ON_INSTRUCTION
